Fanuc TP program (LS listing): HOME_POS_LEFT_SIDE.LS

/PROG  HOME_POS_LEFT_SIDE
/ATTR
OWNER		= MNEDITOR;
COMMENT		= "";
PROG_SIZE	= 497;
CREATE		= DATE 22-06-14  TIME 10:07:14;
MODIFIED	= DATE 25-11-14  TIME 22:02:28;
FILE_NAME	= ;
VERSION		= 0;
LINE_COUNT	= 6;
MEMORY_SIZE	= 845;
PROTECT		= READ_WRITE;
TCD:  STACK_SIZE	= 0,
      TASK_PRIORITY	= 50,
      TIME_SLICE	= 0,
      BUSY_LAMP_OFF	= 0,
      ABORT_REQUEST	= 0,
      PAUSE_REQUEST	= 0;
DEFAULT_GROUP	= 1,*,*,*,*;
CONTROL_CODE	= 00000000 00000000;
LOCAL_REGISTERS	= 0,0,0;
/MN
   1:  UFRAME_NUM=1 ;
   2:  UTOOL_NUM=1 ;
   3:   ;
   4:J P[1] 100% FINE    ;
   5:   ;
   6:  WAIT DO[20:HOME_POSITION_LEFT]=ON    ;
/POS
P[1]{
   GP1:
	UF : 1, UT : 1,
	J1=    40.224 deg,	J2=   140.548 deg,	J3=   -35.409  mm,
	J4=  -180.772 deg
};
/END
